Staubli VAL3: getListItem.pgx

public program getListItem(string& x_sItem[] (dimensions=1), num x_nIndex (dimensions=1))
  local trsf l_tTrsf
  local string l_sItem[6]
  local string l_sEvent
begin
  //
  // define the item to show in the edit page Traj
  // customize an array and copy to x_sItem...
  //
  // see other traj as example
  // 0 > appro
  // 1 > point
  // 2 > depart
  // take it
  switch pEditPoint.tData[x_nIndex].nType
    case 0
      l_sEvent="appro  "
    break
    case 1
      l_sEvent="coord  "
    break
    case 2
      l_sEvent="depart "
    break
  endSwitch
  l_tTrsf=pEditPoint.tData[x_nIndex].pPoint.trsf
  // show them
  l_sItem[0]=(l_sEvent+" X > "+toString(".2",l_tTrsf.x))
  l_sItem[1]=(l_sEvent+" Y > "+toString(".2",l_tTrsf.y))
  l_sItem[2]=(l_sEvent+" Z > "+toString(".2",l_tTrsf.z))
  l_sItem[3]=(l_sEvent+"RX > "+toString(".2",l_tTrsf.rx))
  l_sItem[4]=(l_sEvent+"RY > "+toString(".2",l_tTrsf.ry))
  l_sItem[5]=(l_sEvent+"RZ > "+toString(".2",l_tTrsf.rz))
  // look for intermediate point
  call use:stringCopy(l_sItem,x_sItem)
end
